(*			
	RafalOS
	Rafał Osajda		22.12.2025		TC 4024.66
	Interejs łączacy kilka 
*)
INTERFACE ITF_Component1_HMI_Connector EXTENDS 
	ITF_BaseComponent_HMI_Connector, ITF_Component1_HMI_Connector_View, ITF_Component1_HMI_Connector_Command

END_INTERFACE

(* stored: Version 1.1.0.1
   Itf ITF_Component1_HMI_Connector: Id {65cc0835-fef4-0d15-03a3-f2012ec27258} *)
